		(* ---------------------- Debug-Message ----------------------------*)
		(*IF _debug_enable THEN
			LOG_CL.NEW_MSG := 'FS: File_Start Mode=~1';
			LOG_CL.PRINTF[1] := BYTE_TO_STRING(FSD.MODE);
			LOG_MSG();
		END_IF;*)
		(* -----------------------------------------------------------------------------*)

		(* Initialisierung *)
		X.sNetId := '';
		X.tTimeout := T#5s;
		X.nPort := 10000; (* AMSPORT_R3_SYSSERV *)

		buf_size := SIZEOF(PT.BUFFER);
		close_time := T#1ms; (* wenn Schritt aktiv ist, dann Close-Timer rücksetzen *)

		IF FSD.MODE = 4 THEN (* File_Remove *)
			IF handle > 0 THEN
				File_change := TRUE;
				step := 32000; (* File_Close ausführen *)
			ELSE
				step := 90; (* File_Remove ausführen *)
			END_IF;

		ELSIF FSD.MODE = 5 THEN (* File_Close *)
			step := 32000; (* File_Close ausführen *)

		ELSIF handle = 0 THEN (* MODE 1,2,3 *)
			step := 100; (* File muss erst geöffnet werden *)

		ELSE (* File ist geöffnset *)
			IF used_filename = FSD.FILENAME AND FSD.MODE = last_mode THEN (* kein Moduswechsel ? *)
				step := 200; (* ohne open prozedure weitermachen *)
			ELSE
				step := 32000;
				File_change := TRUE;
			END_IF;
		END_IF;

	ELSIF handle > 0 THEN (* offene Datei gefunden - AutoClose Modus *)
		IF FSD.AUTO_CLOSE > T#0s THEN
			close_time := close_time + t_diff; (* Close_Time hochzählen *)
			IF close_time > FSD.AUTO_CLOSE THEN (* Zeit überschrittenen *)
				step := 32000; (* automatisch Datei schliessen *)
			END_IF;
		END_IF;
	END_IF;

(* ----------------------------------- *)
090: (* File_Remove *)
	command := 7; (* File Remove *)
	step := 95;

095: (* File_Remove beendet *)
	IF command = 0 THEN
		step := 30000; (* Beenden *)
	END_IF;
(* ----------------------------------- *)

100: (* File_Open *)
	IF FSD.MODE = 3 THEN (* Open_New + File Write *)
		open_mode := 16#0001_001A; (* PATH_GENERIC + WRITEPLUS + BINARY *)
	ELSE (* Mode 1 Open_Exist + File _Read / Mode 2 Open_Exist + File_Write *)
		open_mode := 16#0001_0019; (* PATH_GENERIC + READPLUS + BINARY *)
	END_IF;
	command := 1; (* FileOpen *)
	step := 105;

105: (* File Open beendet *)
	IF command = 0 THEN
		IF error THEN
			step := 30000; (* Beenden *)
		ELSE
			(* Filedaten eintragen *)
			close_time := T#1ms; (* Timer freigeben *)
			handle := open_handle;
			used_filename := FSD.FILENAME;
			file_position := UDINT#4294967295; (* maximal = unbekannt *)
			last_mode := FSD.MODE;
			step := 110;
		END_IF;
	END_IF;

110: (* File Seek *)
	command := 5; (* File-Seek *)
	seek_position := 0;
	seek_mode := 2; (* SEEK_END - Seek from the end of file *)
	step := 115;

115: (* File Seek beendet *)
	IF command = 0 THEN
		IF error THEN
			step := 30000; (* Beenden *)
		ELSE
			command := 6; (* File-Tell starten *)
			step := 120;
		END_IF;
	END_IF;

120: (* File Tell beendet *)
	IF command = 0 THEN
		IF error THEN
			step := 30000; (* Beenden *)
		ELSE
			FSD.FILE_SIZE := tell_position; (* aktuelle Dateigroesse *)
			FSD.FILE_OPEN := TRUE;
			step := 200;
		END_IF;
	END_IF;

200: (* File Seek *)
	IF FSD.OFFSET > FSD.FILE_SIZE THEN (* prüfe auf gültige offset-vorgabe *)
		error_code := 255;
		step := 30000; (* Beenden *)
	ELSIF FSD.OFFSET <> file_position THEN
		command := 5; (* File-Seek *)
		seek_position := FSD.OFFSET;
		seek_mode := 0; (* Seek from beginning of file *)
		step := 210;
	ELSE
		step := 300;
	END_IF;

210: (* File Seek *)
	IF command = 0 THEN
		file_position := seek_position;
		IF error THEN
			step := 30000; (* Beenden *)
		ELSE
			step := 300;
		END_IF;
	END_IF;

300: (* Read or Write ? *)
	IF FSD.MODE = 1 THEN
		step := 400; (* Read *)
	ELSE
		step := 500; (* Write *)
	END_IF;

400: (* File Read *)
	IF UINT_TO_UDINT(PT.SIZE) > buf_size THEN (* Leselänge auf Buffergroesse begrenzen *)
		read_max_length := buf_size;
	ELSE
		read_max_length := UINT_TO_UDINT(PT.SIZE);
	END_IF;

	IF read_max_length > buf_size THEN
		read_max_length := buf_size;  (* Leselänge auf Buffergroesse begrenzen *)
	END_IF;

	(* Leselänge an Dateilänge anpassen *)
	IF file_position + read_max_length > FSD.FILE_SIZE THEN
		read_max_length := FSD.FILE_SIZE - file_position;
	END_IF;

	IF read_max_length > 0 THEN
		command := 3; (* File_Read *)
		step := 410;
	ELSE
		PT.SIZE := UINT#0;
		step := 30000; (* Beenden *)
	END_IF;

410: (* File Read *)
	IF command = 0 THEN
		PT.SIZE := UDINT_TO_UINT(length_read);
		IF NOT Error THEN
			file_position := file_position + length_read; (* aktueller File_Position korrigieren *)
			FSD.OFFSET := file_position;
		END_IF;
		step := 30000; (* Beenden *)
	END_IF;

500: (* File Write *)
	IF UINT_TO_UDINT(PT.SIZE) > buf_size THEN (* Schreiblänge auf Buffergroesse begrenzen *)
		write_length := buf_size;
	ELSE
		write_length := UINT_TO_UDINT(PT.SIZE);
	END_IF;

	IF write_length > 0 THEN
		command := 4; (* File_Write *)
		step := 510;
	ELSE
		step := 30000; (* Beenden *)
	END_IF;

510:
	IF command = 0 THEN
		IF NOT Error THEN
			file_position := file_position + length_written; (* aktueller File_Position korrigieren *)
			FSD.OFFSET := file_position;
			IF file_position > FSD.FILE_SIZE THEN (* Datei ist groesser geworden *)
				FSD.FILE_SIZE := file_position;
			END_IF;
		END_IF;
		step := 30000; (* Beenden *)
	END_IF;

 (* --------------------------------------------- *)

30000: (* Befehl fertig *)
	FSD.MODE := 0;
	FSD.ERROR := error_code;
	step := 0;

	(* ---------------- Debug-Message -----------------------*)
	(*IF _debug_enable THEN
		LOG_CL.NEW_MSG := 'FS: File_Stop: File ~1, error ~7, code ~8';
		LOG_CL.PRINTF[1]  := used_filename;
		LOG_CL.PRINTF[7]  := INT_TO_STRING(BOOL_TO_INT(error));
		LOG_CL.PRINTF[8]  := BYTE_TO_STRING(error_code);
		LOG_MSG();
	END_IF;*)
	(* --------------------------------------------- *)

32000:
	close_time := T#0s; (* Timer stoppen *)
	IF handle > 0 THEN
		command := 2; (* File_Close ausführen *)
	END_IF;
	step := 32100;

32100:
	IF command = 0 THEN (* File Close beendet *)
		(* Filedaten ablöschen *)
		FSD.FILE_OPEN := FALSE;
		file_position := 0;
		FSD.FILE_SIZE := 0;
		FSD.OFFSET := 0;
		used_filename := '';
		handle := 0;

		(* File_Name wurde fliegend geändert ? *)
		IF file_change THEN
			file_change := FALSE;
			step := 0;
		ELSE
			step := 30000;
		END_IF;
	END_IF;

END_CASE;

(* 1 = file_open
   2 = file_close
   3 = file_read
   4 = file_write
   5 = file_seek
   6 = file_tell
   7 = file_remove
*) 

X(bExecute := FALSE); (* Zyklischer FW_AdsRdWrt Aufruf *)

(* ------------ File Open ------------- *)
IF command = 1 THEN
	IF NOT para THEN
		para := TRUE;
		X(	nIdxGrp := 120, (* SYSTEMSERVICE_FOPEN *)
			nidxOffs := open_mode,
			cbWriteLen := SIZEOF(FSD.FILENAME),
			pWriteBuff := ADR(FSD.FILENAME),
			cbReadLen := SIZEOF(tmpDW),
			pReadBuff := ADR(tmpDW),
			bExecute := TRUE
			);
	ELSIF X.bBusy = FALSE THEN
		para := FALSE;
		error := X.bError;
		error_code := SEL(error,0,UDINT_TO_BYTE(X.nErrId + 16#10));

		IF X.cbRead >= SIZEOF(tmpDW) THEN
			open_handle := UDINT_TO_UINT(tmpDW);
		ELSE
			open_handle := 0;
		END_IF;
		command := 0;

		(* ---------------- Debug-Message -----------------------*)
		(*IF _debug_enable THEN
			LOG_CL.NEW_MSG := 'FS: Open: File ~1, handle ~2 , mode ~3 , error ~7, code ~8';
			LOG_CL.PRINTF[1] := FSD.FILENAME;
			LOG_CL.PRINTF[2] := DWORD_TO_STRING(open_handle);
			LOG_CL.PRINTF[3] := DWORD_TO_STRING(open_mode);
			LOG_CL.PRINTF[7] := INT_TO_STRING(BOOL_TO_INT(error));
			LOG_CL.PRINTF[8] := BYTE_TO_STRING(error_code);
			LOG_MSG();
		END_IF;*)
		(* -----------------------------------------------------------------*)
	END_IF;
END_IF;

(* ----------- File Close ------------- *)
IF command = 2 THEN
	IF NOT para THEN
		para := TRUE;
		X(	nIdxGrp := 121, (* SYSTEMSERVICE_FCLOSE *)
			nidxOffs := handle,
			cbWriteLen := 0,
			pWriteBuff := 0,
			cbReadLen := 0,
			pReadBuff := 0,
			bExecute := TRUE
			);
	ELSIF X.bBusy = FALSE THEN
		para := FALSE;
		error := X.bError;
		error_code := SEL(error,0,UDINT_TO_BYTE(X.nErrId + 16#30));
		command := 0;
		(* ---------------- Debug-Message -----------------------*)
		(*IF _debug_enable THEN
			LOG_CL.NEW_MSG := 'FS: Close: File ~1, error ~7, code ~8';
			LOG_CL.PRINTF[1] := used_filename;
			LOG_CL.PRINTF[7] := INT_TO_STRING(BOOL_TO_INT(error));
			LOG_CL.PRINTF[8] := BYTE_TO_STRING(error_code);
			LOG_MSG();
		END_IF;*)
		(* -----------------------------------------------------------------*)
	END_IF;
END_IF;

(* ------------ File Read ------------- *)
IF command = 3 THEN
	IF NOT para THEN
		para := TRUE;
		X(	nIdxGrp := 122, (* SYSTEMSERVICE_FREAD *)
			nidxOffs := handle,
			cbWriteLen := 0,
			pWriteBuff := 0,
			cbReadLen := read_max_length,
			pReadBuff := ADR(PT.BUFFER),
			bExecute := TRUE
			);
	ELSIF X.bBusy = FALSE THEN
		length_read := X.cbRead;
		para := FALSE;
		error := X.bError;
		error_code := SEL(error,0,UDINT_TO_BYTE(X.nErrId + 16#40));
		command := 0;

		(* ---------------- Debug-Message -----------------------*)
		(*IF _debug_enable THEN
			LOG_CL.NEW_MSG := 'FS: Read: File ~1, soll ~2,ist ~3 ,error ~7, code ~8';
			LOG_CL.PRINTF[1] := used_filename;
			LOG_CL.PRINTF[2] := UDINT_TO_STRING(read_max_length);
			LOG_CL.PRINTF[3] := UDINT_TO_STRING(length_read);
			LOG_CL.PRINTF[7] := INT_TO_STRING(BOOL_TO_INT(error));
			LOG_CL.PRINTF[8] := BYTE_TO_STRING(error_code);
			LOG_MSG();
		END_IF;*)
		(* -----------------------------------------------------------------*)
	END_IF;
END_IF;

(* ------------ File Write ------------- *)
IF command = 4 THEN
	IF NOT para THEN
		para := TRUE;
		X(	nIdxGrp := 123, (* SYSTEMSERVICE_FWRITE *)
			nidxOffs := handle,
			cbWriteLen := write_length,
			pWriteBuff := ADR(PT.BUFFER),
			cbReadLen := SIZEOF(length_written),
			pReadBuff := ADR(length_written),
			bExecute := TRUE
			);
	ELSIF X.bBusy = FALSE THEN
		para := FALSE;
		error := X.bError;
		error_code := SEL(error,0,UDINT_TO_BYTE(X.nErrId + 16#50));
		command := 0;

		(* ---------------- Debug-Message -----------------------*)
		(*IF _debug_enable THEN
			LOG_CL.NEW_MSG := 'FS: Write: File ~1, soll ~2,ist ~3 ,error ~7, code ~8';
			LOG_CL.PRINTF[1] := used_filename;
			LOG_CL.PRINTF[2] := UDINT_TO_STRING(write_length);
			LOG_CL.PRINTF[3] := UDINT_TO_STRING(length_written);
			LOG_CL.PRINTF[7] := INT_TO_STRING(BOOL_TO_INT(error));
			LOG_CL.PRINTF[8] := BYTE_TO_STRING(error_code);
			LOG_MSG();
		END_IF;*)
		(* -----------------------------------------------------------------*)
	END_IF;
END_IF;

(* ------------ File Seek ------------- *)
IF command = 5 THEN
	IF NOT para THEN
		para := TRUE;
		seek_data[0] := UDINT_TO_DINT(seek_position);
		seek_data[1] := INT_TO_DINT(seek_mode);

		X(	nIdxGrp := 124, (* SYSTEMSERVICE_FSEEK *)
			nidxOffs := handle,
			cbWriteLen := SIZEOF(seek_data),
			pWriteBuff := ADR(seek_data),
			cbReadLen := 0,
			pReadBuff := 0,
			bExecute := TRUE
			);
	ELSIF X.bBusy = FALSE THEN
		para := FALSE;
		error := X.bError;
		error_code := SEL(error,0,UDINT_TO_BYTE(X.nErrId + 16#60));
		command := 0;

		(* ---------------- Debug-Message -----------------------*)
		(*IF _debug_enable THEN
			LOG_CL.NEW_MSG := 'FS: Seek: File ~1,pos ~3 ,error ~7, code ~8';
			LOG_CL.PRINTF[1] := used_filename;
			LOG_CL.PRINTF[3] := UDINT_TO_STRING(seek_position);
			LOG_CL.PRINTF[7] := INT_TO_STRING(BOOL_TO_INT(error));
			LOG_CL.PRINTF[8] := BYTE_TO_STRING(error_code);
			LOG_MSG();
		END_IF;*)
		(* -----------------------------------------------------------------*)
	END_IF;
END_IF;

(* ------------ File Tell ------------- *)
IF command = 6 THEN
	IF NOT para THEN
		para := TRUE;
		X(	nIdxGrp := 125, (* SYSTEMSERVICE_FTELL *)
			nidxOffs := handle,
			cbWriteLen := 0,
			pWriteBuff := 0,
			cbReadLen := SIZEOF(tell_position),
			pReadBuff := ADR(tell_position),
			bExecute := TRUE
			);
	ELSIF X.bBusy = FALSE THEN
		para := FALSE;
		error := X.bError;
		error_code := SEL(error,0,UDINT_TO_BYTE(X.nErrId + 16#70));
		command := 0;

		(* ---------------- Debug-Message -----------------------*)
		(*IF _debug_enable THEN
			LOG_CL.NEW_MSG := 'FS: Tell: File ~1, pos ~3 ,error ~7, code ~8';
			LOG_CL.PRINTF[1] := used_filename;
			LOG_CL.PRINTF[3] := UDINT_TO_STRING(tell_position);
			LOG_CL.PRINTF[7] := INT_TO_STRING(BOOL_TO_INT(error));
			LOG_CL.PRINTF[8] := BYTE_TO_STRING(error_code);
			LOG_MSG();
		END_IF;*)
		(* -----------------------------------------------------------------*)
	END_IF;
END_IF;

(* ------------ File Remove ------------- *)
IF command = 7 THEN
	IF NOT para THEN
		para := TRUE;
		X(	nIdxGrp := 131, (* SYSTEMSERVICE_FDELETE *)
			nidxOffs := 16#0001_0000, (* PATH_GENERIC *)
			cbWriteLen := SIZEOF(FSD.FILENAME),
			pWriteBuff := ADR(FSD.FILENAME),
			cbReadLen := 0,
			pReadBuff := 0,
			bExecute := TRUE
			);
	ELSIF X.bBusy = FALSE THEN
		para := FALSE;
		error := X.bError;
		error_code := SEL(error,0,UDINT_TO_BYTE(X.nErrId + 16#80));
		command := 0;

		(* ---------------- Debug-Message -----------------------*)
		(*IF _debug_enable THEN
			LOG_CL.NEW_MSG := 'FS: Remove: File ~1, error ~7, code ~8';
			LOG_CL.PRINTF[1] := FSD.FILENAME;
			LOG_CL.PRINTF[7] := INT_TO_STRING(BOOL_TO_INT(error));
			LOG_CL.PRINTF[8] := BYTE_TO_STRING(error_code);
			LOG_MSG();
		END_IF;*)
		(* -----------------------------------------------------------------*)
	END_IF;
END_IF;

(* ---------------- Debug-Message -----------------------*)
(*IF _debug_enable THEN
	IF step_last <> step THEN
		LOG_CL.NEW_MSG := 'FS: Step: ~1';
		LOG_CL.PRINTF[1] := INT_TO_STRING(step);
		LOG_MSG();
	END_IF;
	step_last := step;
END_IF;*)
(* -----------------------------------------------------------------*)

(* revision history
ks	23. sep. 2010	rev 1.0
	original version
*)

END_FUNCTION_BLOCK

// ---- oscat_network/POUs/HARDWARE/IP_CONTROL_RESET_1.TcPOU
FUNCTION_BLOCK IP_CONTROL_RESET_1
VAR_INPUT
END_VAR
VAR_OUTPUT
	READY : BOOL;
END_VAR
VAR
	fbSocketCloseAll : FB_SocketCloseAll;
	step : BYTE;
END_VAR

(* On PLC reset or program download close all old connections *)

CASE TCP_SERVER_RESET OF

2:	READY := TRUE;
	RETURN;

1:	IF step = 0 THEN
		RETURN;
	END_IF;

0:	TCP_SERVER_RESET := 1; (* Reset ist aktiv *)
	step := 1;

END_CASE;

CASE step OF

0:	RETURN;

1:	fbSocketCloseAll(sSrvNetId:= '', bExecute:= TRUE, tTimeout:= T#10s );
	step := 2;

2:	fbSocketCloseAll(bExecute:= FALSE);
	IF fbSocketCloseAll.bBusy = FALSE THEN
		step := 0;
		TCP_SERVER_RESET := 2; (* Reset durchgeführt , Bereit zur Verwendung *)
	END_IF;

END_CASE;

END_FUNCTION_BLOCK

// ---- oscat_network/POUs/OTHER/NETWORK_VERSION.TcPOU
FUNCTION NETWORK_VERSION : DWORD
VAR_INPUT
	IN : BOOL;
END_VAR

(*
version 1.0	02. feb 2011
programmer 	kst
tested by		oscat

network_version returns the version number in dword format
110 is library version 1.10
if IN = true, the release date will be returned

*)

IF in THEN
	NETWORK_VERSION := DATE_TO_DWORD(D#2011-12-01);
ELSE
	NETWORK_VERSION := 121;
END_IF;

(* revision history
ks	2. feb 2011	rev 1.0
	original version

*)

END_FUNCTION

// ---- oscat_network/POUs/TELNET_VISION/TN_SC_READ_ATTR.TcPOU
FUNCTION_BLOCK TN_SC_READ_ATTR
VAR
	in_Offset : INT;
END_VAR
VAR_INPUT
	Iin_Y : INT;
	Iin_X : INT;
END_VAR
VAR_OUTPUT
	Oby_ATTR : BYTE;
END_VAR
VAR_IN_OUT
	Xus_TN_SCREEN : us_TN_SCREEN;
END_VAR

(*
version 1.0		10. mai 2010
programmer		ks
tested by		ks

TN_SC_READ_ATTR gibt den Farbcode einer Koordinate vom Bildschirm aus

*)

IF TN_SC_XY_ERROR(Iin_X,Iin_Y) THEN RETURN; END_IF;
in_Offset := (Iin_Y * 80) + Iin_X;
Oby_ATTR := Xus_TN_SCREEN.bya_COLOR[in_Offset]; (* Attribute auslesen *)

(* revision history
ks	10. mai. 2010	rev 1.0
	original version
*)

END_FUNCTION_BLOCK

// ---- oscat_network/POUs/TELNET_VISION/TN_SC_READ_CHAR.TcPOU
FUNCTION_BLOCK TN_SC_READ_CHAR
VAR
	in_Offset : INT;
END_VAR
VAR_INPUT
	Iin_Y : INT;
	Iin_X : INT;
END_VAR
VAR_OUTPUT
	Oby_CHAR : BYTE;
END_VAR
VAR_IN_OUT
	Xus_TN_SCREEN : us_TN_SCREEN;
END_VAR

(*
version 1.0		10. mai 2010
programmer		ks
tested by		ks

TN_SC_READ_CHAR gibt das Zeichen einer Koordinate vom Bildschirm aus
*)

IF TN_SC_XY_ERROR(Iin_X,Iin_Y) THEN RETURN; END_IF;
in_Offset := (Iin_Y * 80) + Iin_X;
Oby_CHAR := Xus_TN_SCREEN.bya_CHAR[in_Offset]; (* Charakter auslesen *)

(* revision history
ks	10. mai. 2010	rev 1.0
	original version
*)

END_FUNCTION_BLOCK

// ---- oscat_network/POUs/TELNET_VISION/TN_SC_WRITE_ATTR.TcPOU
FUNCTION_BLOCK TN_SC_WRITE_ATTR
VAR
	in_Offset : INT;
END_VAR
VAR_INPUT
	Iin_Y : INT;
	Iin_X : INT;
	Iby_ATTR : BYTE;
END_VAR
VAR_IN_OUT
	Xus_TN_SCREEN : us_TN_SCREEN;
END_VAR

(*
version 1.0		10. mai 2010
programmer		ks
tested by		ks

TN_SC_WRITE_ATTR ändert an der angegebenen Koordinate den Farbcode
*)

IF TN_SC_XY_ERROR(Iin_X,Iin_Y) THEN RETURN; END_IF;
in_Offset := (Iin_Y * 80) + Iin_X;
Xus_TN_SCREEN.bya_COLOR[in_Offset] := Iby_ATTR; (* Attribute schreiben *)

(* revision history
ks	10. mai. 2010	rev 1.0
	original version
*)

END_FUNCTION_BLOCK

// ---- oscat_network/POUs/TELNET_VISION/TN_SC_WRITE_CHAR.TcPOU
FUNCTION_BLOCK TN_SC_WRITE_CHAR
VAR
	in_Offset : INT;
END_VAR
VAR_INPUT
	Iin_Y : INT;
	Iin_X : INT;
	Iby_CHAR : BYTE;
END_VAR
VAR_IN_OUT
	Xus_TN_SCREEN : us_TN_SCREEN;
END_VAR

(*
version 1.0		10. mai 2010
programmer		ks
tested by		ks

TN_SC_WRITE_CHAR schreibt ein einzelnes Zeichen an die angegebenen Koordinate ohne den vorhandenen Farbcode zu ändern 
*)

IF TN_SC_XY_ERROR(Iin_X,Iin_Y) THEN RETURN; END_IF;
in_Offset := (Iin_Y * 80) + Iin_X;
Xus_TN_SCREEN.bya_CHAR[in_Offset] := Iby_CHAR; (* Charakter schreiben *)

(* revision history
ks	10. mai. 2010	rev 1.0
	original version
*)

END_FUNCTION_BLOCK

// ---- oscat_network/POUs/TELNET_VISION/TN_SC_WRITE_EOS.TcPOU
FUNCTION_BLOCK TN_SC_WRITE_EOS
VAR
	TN_SC_WRITE : TN_SC_WRITE;
END_VAR
VAR_INPUT
	Iby_ATTR : BYTE;
	Ist_STRING : STRING;
END_VAR
VAR_IN_OUT
	Xus_TN_SCREEN : us_TN_SCREEN;
END_VAR

(*
version 1.0		10. mai 2010
programmer		ks
tested by		ks

TN_SC_WRITE_EOS schreibt einem Text an das Ende des zuletzt geschreibene Texts 
*)

TN_SC_WRITE(Iin_Y := Xus_TN_SCREEN.in_EOS_Offset / 80, (* aktuelle Zeile ausrechnen *)
			Iin_X := Xus_TN_SCREEN.in_EOS_Offset MOD 80, (* aktuelle Spalte ausrechnen *)
			Iby_ATTR := Iby_ATTR,
			Ist_STRING := Ist_STRING,
			Xus_TN_SCREEN := Xus_TN_SCREEN);

(* revision history
ks	10. mai. 2010	rev 1.0
	original version
*)

END_FUNCTION_BLOCK

// ---- oscat_network/POUs/WEATHER/MOON_PHASE.TcPOU
FUNCTION_BLOCK MOON_PHASE
VAR_INPUT
	XDT : DT;
	SCALE : BYTE := 12;
	UPDATE : TIME := T#1h;
END_VAR
VAR_OUTPUT
	PHASE : BYTE;
END_VAR
VAR
	x : UDINT;
	last_dt : DT;
END_VAR

(*
version 1.0		15. may. 2011
programmer		ks
tested by			ks

MOON_PHASE berechnet die aktuelle Mondphase
*)

IF XDT - last_dt > UPDATE THEN
	x := (DT_TO_UDINT(XDT) - 603240) MOD 2551392;
	PHASE := UDINT_TO_BYTE(SCALE * x / 2551392) ;
	last_dt := XDT;
END_IF;

(* revision history
ks	15.may. 2011	rev 1.0
	original version

*)

END_FUNCTION_BLOCK
